FUNCTION_BLOCK TcoObjectEqualsTest EXTENDS TcoCore.TcoObject
VAR
    _someNumber : INT;
    _someString : STRING;
END_VAR

METHOD PUBLIC EqualsTo : BOOL
VAR_INPUT
    Object : ITcoObject;
END_VAR
VAR
    _object : POINTER TO TcoObjectEqualsTest;
END_VAR
IF (__QUERYPOINTER(Object, _object)) THEN
    EqualsTo := _object^._someNumber = THIS^._someNumber AND _object^._someString = THIS^._someString;
END_IF;
END_METHOD

PROPERTY SomeNumber : INT
GET
SomeNumber := _someNumber;
END_GET
SET
_someNumber := SomeNumber;
END_SET
END_PROPERTY

PROPERTY SomeString : STRING
GET
SomeString := _someString;
END_GET
SET
_someString := SomeString;
END_SET
END_PROPERTY

END_FUNCTION_BLOCK

(* stored: Version 1.1.0.1
   POU TcoObjectEqualsTest: Id {95fdb37c-6061-07da-0252-b29845f7825c}, SpecialFunc None
   Method EqualsTo: Id {25ebe5f5-998c-0972-08b6-13a507a3c4f7}
   Property SomeNumber: Id {d3dac4aa-994e-0f33-0e8b-69c000edb619}
   Get Get: Id {d8dc5e21-4199-01af-2f1d-61e8d681824b}
   Set Set: Id {4128da7d-65d5-0a2f-23ba-beceb619dc5d}
   Property SomeString: Id {60bdc7e9-443a-055d-05af-bc5b993e9510}
   Get Get: Id {4b0df5d1-9706-0d1a-1ebe-34fb209ab266}
   Set Set: Id {a3a5d345-3fbb-093f-3b2e-fb9738048b57} *)
